Universal Robots URScript: UR.script

def test1():
  set_standard_analog_input_domain(0, 1)
  set_standard_analog_input_domain(1, 1)
  set_tool_analog_input_domain(0, 1)
  set_tool_analog_input_domain(1, 1)
  set_analog_outputdomain(0, 0)
  set_analog_outputdomain(1, 1)
  set_tool_voltage(12)
  set_input_actions_to_default()
  set_tool_digital_input_action(0, "freedrive")
  set_tcp(p[0.0,0.0,0.0,0.0,0.0,0.0])
  set_payload(0.0)
  set_gravity([0.0, 0.0, 9.82])
  global plane=p[0.26223651820150723,-0.2742010986097009,0.3630950575382667,1.4903437393745607,0.586436574758555,0.5866887336171906]
  global rot0=p[0.2622439651785617,-0.27422233482255337,0.3631149856628333,1.49024657548656,0.5863547897330073,0.5865270767774048]
  global rot30=p[0.2622792129724982,-0.2741385033679078,0.36312411214661144,1.1310116437705044,1.0907043746297485,-0.02761348091861309]
  global u28857_7=p[0.26223651820150723,-0.2742010986097009,0.3630950575382667,-0.49861789472297735,1.7850505161549586,-1.5188003198916027]
  global u28857_8=p[0.26223158448185935,-0.2742473640182322,0.4998711637170484,-0.49871852205459943,1.7850442858255617,-1.5187642847920932]
  global u28857_9=p[0.39987620742062946,-0.14601257038822735,0.500103831966284,-0.4613436824347936,1.8067330112900566,-1.5494011717976852]
  while (True):
    $ 1 "机器人程序"
    $ 2 "MoveJ"
    $ 3 "路点_1"
    movej([2.5888870422118337, -2.0982167357949173, -1.3630170810218054, 0.565982974356273, 1.392352124990663, 0.059640793444356355], a=1.0471975511965976, v=0.08726646259971647, r=0.01)
    $ 4 "路点_2"
    movej([2.5970970573705854, -2.09845147161629, -1.6394005772306208, 0.4315635635154322, 1.4514542711307294, 0.059725258499383926], a=1.0471975511965976, v=0.08726646259971647, r=0.01)
    $ 5 "路点_3"
    movej([2.899465594800887, -2.098189655934469, -1.4078483950635494, 0.3242074251174927, 1.3993344931054166, 0.2700585346200387], a=1.0471975511965976, v=0.08726646259971647, r=0.01)
    $ 6 "路点_4"
    movej([2.8227407932281494, -2.0876431048126047, -1.0814397970782679, 0.49084239972382804, 1.3659042794725975, 0.27261080157430845], a=1.0471975511965976, v=0.08726646259971647, r=0.01)
  end
end
